// TIA Portal V19 export
FUNCTION_BLOCK "PathTest"   // FB135, LAD
// stored: Access Published, MemoryReserve 100, SetENOAutomatically false
   VAR_INPUT
      AreaInterface : "AreaInterface";
      DevicesInSafeState : Bool;   // Axis in safe state
      Door_OK : Bool;   // All door of axis device ok
   END_VAR
   VAR_OUTPUT
      AlarmPresence : Bool;   // Cumulative alarm presence
      WarningPresence : Bool;   // Cumulative warning presence
      DriveCtrlSafe : Bool;   // Safe ctrl for enable axis drive
   END_VAR
   VAR_IN_OUT
      PathTest : "PathTestSignal";
   END_VAR
   VAR
      Alarm : Struct
         TestTimeout : Bool;
      END_STRUCT;
      Warning : Struct
         TestRequired : Bool;
         MaxRetry : Bool;
      END_STRUCT;
      HMI : "PathTestHMI";
      Timeout : IEC_TIMER;
      TimeBetweenRetry : IEC_TIMER;
      Retry_PEAux : Bool;
      Retry : UInt;
   END_VAR
   VAR_TEMP
      Man_Start : Bool;
      Auto_Start : Bool;
   END_VAR
   VAR CONSTANT
      MAX_RETRY : UInt := 3;
   END_VAR
   VAR_TEMP   // added for the SCL form of the ladder/FBD networks
      _w1 : Bool;
   END_VAR
BEGIN

REGION Network 1: Warning: Path Test Necessary
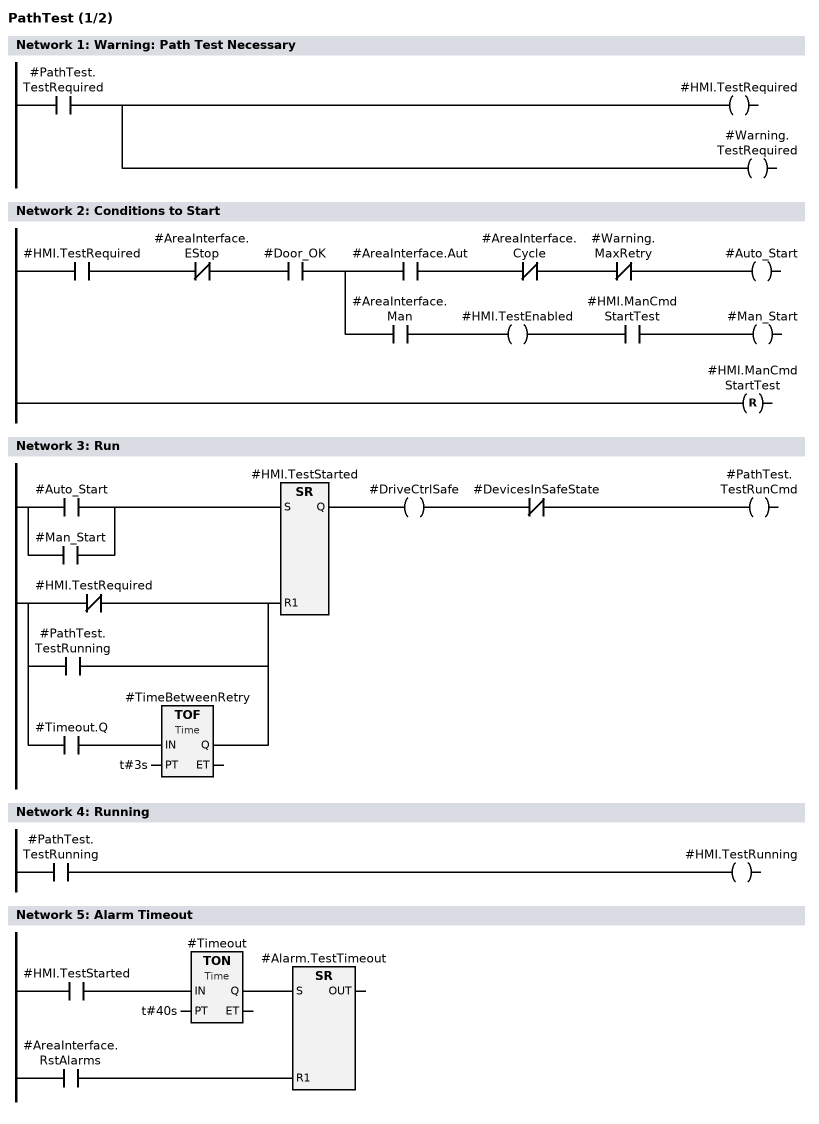
   RUNG wire#powerrail
      Contact( #PathTest.TestRequired )
      wire#w1
      Coil( #HMI.TestRequired )
   END_RUNG
   RUNG wire#w1
      Coil( #Warning.TestRequired )
   END_RUNG
   // the same network as SCL:
   #HMI.TestRequired := #PathTest.TestRequired;
   #Warning.TestRequired := #PathTest.TestRequired;
END_REGION

REGION Network 2: Conditions to Start
   RUNG wire#powerrail
      Contact( #HMI.TestRequired )
      I_Contact( #AreaInterface.EStop )
      Contact( #Door_OK )
      wire#w1
      Contact( #AreaInterface.Aut )
      I_Contact( #AreaInterface.Cycle )
      I_Contact( #Warning.MaxRetry )
      Coil( #Auto_Start )
   END_RUNG
   RUNG wire#w1
      Contact( #AreaInterface.Man )
      Coil( #HMI.TestEnabled )
      Contact( #HMI.ManCmdStartTest )
      Coil( #Man_Start )
   END_RUNG
   RUNG wire#powerrail
      R_Coil( #HMI.ManCmdStartTest )
   END_RUNG
   // the same network as SCL:
   #_w1 := #HMI.TestRequired AND NOT #AreaInterface.EStop AND #Door_OK;
   #Auto_Start := #_w1 AND #AreaInterface.Aut AND NOT #AreaInterface.Cycle AND NOT #Warning.MaxRetry;
   #HMI.TestEnabled := #_w1 AND #AreaInterface.Man;
   #Man_Start := #HMI.TestEnabled AND #HMI.ManCmdStartTest;
   #HMI.ManCmdStartTest := FALSE;
END_REGION

REGION Network 3: Run
   RUNG wire#powerrail
      Contact( #Auto_Start )
      wire#w1
      S_SR(operand := #HMI.TestStarted, r1 := wire#w2)
      Coil( #DriveCtrlSafe )
      I_Contact( #DevicesInSafeState )
      Coil( #PathTest.TestRunCmd )
   END_RUNG
   RUNG wire#powerrail
      Contact( #Man_Start )
   END_RUNG wire#w1
   RUNG wire#powerrail
      I_Contact( #HMI.TestRequired )
   END_RUNG wire#w2
   RUNG wire#powerrail
      Contact( #PathTest.TestRunning )
   END_RUNG wire#w2
   RUNG wire#powerrail
      Contact( #Timeout.Q )
      { S7_Templates := "time_type := Time" } #TimeBetweenRetry.TOF(pt := t#3s, et =>)
   END_RUNG wire#w2
   // the same network as SCL:
   #TimeBetweenRetry.TOF(IN := #Timeout.Q, PT := t#3s);
   IF #Auto_Start OR #Man_Start THEN
       #HMI.TestStarted := TRUE;   // SR flip-flop
   END_IF;
   IF NOT #HMI.TestRequired OR #PathTest.TestRunning OR #TimeBetweenRetry.Q THEN
       #HMI.TestStarted := FALSE;
   END_IF;
   #DriveCtrlSafe := #HMI.TestStarted;
   #PathTest.TestRunCmd := #HMI.TestStarted AND NOT #DevicesInSafeState;
END_REGION

REGION Network 4: Running
   RUNG wire#powerrail
      Contact( #PathTest.TestRunning )
      Coil( #HMI.TestRunning )
   END_RUNG
   // the same network as SCL:
   #HMI.TestRunning := #PathTest.TestRunning;
END_REGION

REGION Network 5: Alarm Timeout
   RUNG wire#powerrail
      Contact( #HMI.TestStarted )
      { S7_Templates := "time_type := Time" } #Timeout.TON(pt := t#40s, et =>)
      S_SR(operand := #Alarm.TestTimeout, r1 := wire#w1)
   END_RUNG
   RUNG wire#powerrail
      Contact( #AreaInterface.RstAlarms )
   END_RUNG wire#w1
   // the same network as SCL:
   #Timeout.TON(IN := #HMI.TestStarted, PT := t#40s);
   IF #Timeout.Q THEN
       #Alarm.TestTimeout := TRUE;   // SR flip-flop
   END_IF;
   IF #AreaInterface.RstAlarms THEN #Alarm.TestTimeout := FALSE; END_IF;
END_REGION

REGION Network 6: Automatic Retry
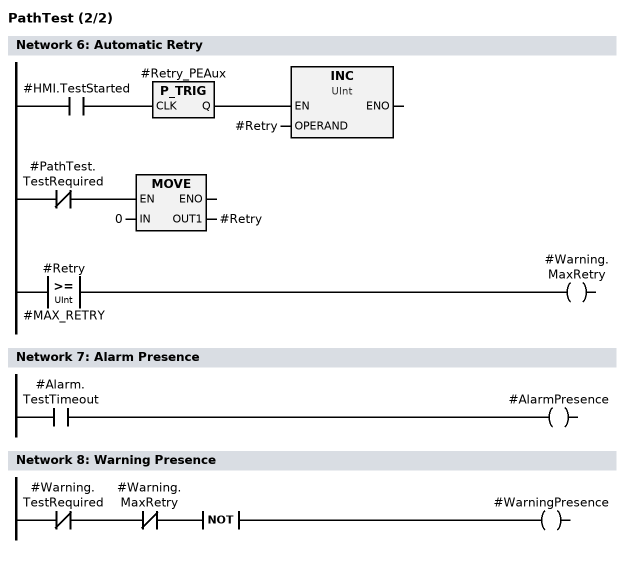
   RUNG wire#powerrail
      Contact( #HMI.TestStarted )
      P_Trig( #Retry_PEAux )
      { S7_Templates := "DestType := UInt" } Inc( #Retry )
   END_RUNG
   RUNG wire#powerrail
      I_Contact( #PathTest.TestRequired )
      Move(in := 0, out1 => #Retry)
   END_RUNG
   RUNG wire#powerrail
      { S7_Templates := "SrcType := UInt" } GE_Contact(in1 := #Retry, in2 := #MAX_RETRY)
      Coil( #Warning.MaxRetry )
   END_RUNG
   // the same network as SCL:
   #_w1 := #HMI.TestStarted AND NOT #Retry_PEAux;   // rising edge
   #Retry_PEAux := #HMI.TestStarted;
   IF #_w1 THEN #Retry := #Retry + 1; END_IF;
   IF NOT #PathTest.TestRequired THEN #Retry := 0; END_IF;
   #Warning.MaxRetry := #Retry >= #MAX_RETRY;
END_REGION

REGION Network 7: Alarm Presence
   RUNG wire#powerrail
      Contact( #Alarm.TestTimeout )
      Coil( #AlarmPresence )
   END_RUNG
   // the same network as SCL:
   #AlarmPresence := #Alarm.TestTimeout;
END_REGION

REGION Network 8: Warning Presence
   RUNG wire#powerrail
      I_Contact( #Warning.TestRequired )
      I_Contact( #Warning.MaxRetry )
      Not()
      Coil( #WarningPresence )
   END_RUNG
   // the same network as SCL:
   #WarningPresence := NOT (NOT #Warning.TestRequired AND NOT #Warning.MaxRetry);
END_REGION
END_FUNCTION_BLOCK
